# EPICS substitutions: vitaraApp/Db/ai_hist_RFChan.substitutions
#
# ai_hist_RFChan.substitutions
#
# Uses the generated ai_hist_pattern.db template
# to create history waveforms for each of the
# specified PV's along with AVG, MAX, MIN,
# RMS, and StdDev for each history.
#
# Required Macros:
#	PV		 - PV name
# Optional Macros:
#	EGU		 - Engineering units, default to ""
#	RMS_LOLO - Low  alarm   limit for $(PV)_RMS, default 0
#	RMS_LOW  - Low  warning limit for $(PV)_RMS, default 0
#	RMS_HIGH - High warning limit for $(PV)_RMS, default 0
#	RMS_HIHI - High alarm   limit for $(PV)_RMS, default 0
#   N_SAMPLES - Number of samples to save in waveforms
# Example
file ai_hist_pattern.db
{
	pattern
	{	PV,						EGU			}
	{	'$(CH)DIODE_PWR',		"V"			}
	{	'$(CH)FEEDBACK_GAIN',	"V"			}
	{	'$(CH)PHASE',			"V"			}
	{	'$(CH)PHASE_X30',		"V"			}
	{	'$(CH)RF_PWR',			"V"			}
}
